(* IEC 61131-3 sources: axopen.integrations.hwc/ctrl/src (part 2) *)

                IF _progress = 452 THEN
                    TaskMessenger.ActivateOnCondition(ULINT#652, _infoTimer.output, eAxoMessageCategory#Warning);
                    IF _infoTimer.output THEN
                        Status.Error.Id := UINT#652;
                    END_IF;

                    IF TRUE THEN
                        _progress := 453;
                    END_IF;
                END_IF;

                IF _progress = 453 THEN
                    TaskMessenger.ActivateOnCondition(ULINT#653, _infoTimer.output, eAxoMessageCategory#Warning);
                    IF _infoTimer.output THEN
                        Status.Error.Id := UINT#653;
                    END_IF;

                    IF TRUE THEN
                        _progress := 454;
                    END_IF;
                END_IF;

                IF _progress = 454 THEN
                    TaskMessenger.ActivateOnCondition(ULINT#654, _infoTimer.output, eAxoMessageCategory#Warning);
                    IF _infoTimer.output THEN
                        Status.Error.Id := UINT#654;
                    END_IF;

                    IF TRUE THEN
                        _progress := 455;
                    END_IF;
                END_IF;

                IF _progress = 455 THEN
                    TaskMessenger.ActivateOnCondition(ULINT#655, _infoTimer.output, eAxoMessageCategory#Warning);
                    IF _infoTimer.output THEN
                        Status.Error.Id := UINT#655;
                    END_IF;

                    IF TRUE THEN
                        _progress := 456;
                    END_IF;
                END_IF;

                IF _progress = 456 THEN
                    TaskMessenger.ActivateOnCondition(ULINT#656, _infoTimer.output, eAxoMessageCategory#Warning);
                    IF _infoTimer.output THEN
                        Status.Error.Id := UINT#656;
                    END_IF;

                    IF TRUE THEN
                        _progress := 457;
                    END_IF;
                END_IF;

                IF _progress = 457 THEN
                    TaskMessenger.ActivateOnCondition(ULINT#657, _infoTimer.output, eAxoMessageCategory#Warning);
                    IF _infoTimer.output THEN
                        Status.Error.Id := UINT#657;
                    END_IF;

                    IF TRUE THEN
                        _progress := 458;
                    END_IF;
                END_IF;

                IF _progress = 458 THEN
                    TaskMessenger.ActivateOnCondition(ULINT#658, _infoTimer.output, eAxoMessageCategory#Warning);
                    IF _infoTimer.output THEN
                        Status.Error.Id := UINT#658;
                    END_IF;

                    IF TRUE THEN
                        _progress := 459;
                    END_IF;
                END_IF;

                IF _progress = 459 THEN
                    TemplateTask_20steps_4.DoneWhen(TRUE);
                END_IF;

                THIS.CallTimers(TRUE);

                TemplateTask_20steps_4.ThrowWhen(_errorTimer.output);
                Status.Action.Id := TO_UINT(_progress);
                TemplateTask_20steps_4.ThrowWhen(StopTask.Duration >= Config.ErrorTime ,'xxxxxxxx');
            END_IF;
            IF TemplateTask_20steps_4.DoneReached() THEN
                Status.Action.Id :=  UINT#241;
                Status.Error.Id :=  UINT#0;
            ELSIF TemplateTask_20steps_4.ErrorOccured() THEN
                Status.Action.Id :=  UINT#940;
                Status.Error.Id  :=  UINT#940;
            ELSIF TemplateTask_20steps_4.AbortTriggered()THEN
                Status.Action.Id :=  UINT#941;
                Status.Error.Id  :=  UINT#941;
            END_IF;
            Messenger.ActivateOnCondition(ULINT#940,TemplateTask_20steps_4.HasError(), eAxoMessageCategory#Error);
            Messenger.ActivateOnCondition(ULINT#941,TemplateTask_20steps_4.IsAborted(), eAxoMessageCategory#Error);
            Messenger.ActivateOnCondition(ULINT#242,TemplateTask_20steps_4.RestoreTriggered() , eAxoMessageCategory#Error);
            IF TemplateTask_20steps_4.RestoreTriggered() AND _progress >= 440 AND _progress <= 459  THEN
                Status.Action.Id :=  UINT#242;
                _progress := 0;
            END_IF;
            //******************************************

            //*************TemplateTask_20steps_5***************
            TemplateTask_20steps_5.SetIsDisabled(FALSE);
            IF TemplateTask_20steps_5.StartTriggered() THEN
                Status.Action.Id :=  UINT#260;
            END_IF;
            Messenger.ActivateOnCondition(ULINT#260,TemplateTask_20steps_5.IsBusy(), eAxoMessageCategory#Info);
            Messenger.ActivateOnCondition(ULINT#261,TemplateTask_20steps_5.IsDone(), eAxoMessageCategory#Info);
            IF TemplateTask_20steps_5.Execute() THEN
                IF _progress = 0 THEN
                    Status.Error.Id := UINT#0;
                    TaskMessenger.Restore();
                    THIS.CallTimers(FALSE);
                    _progress := 460;
                END_IF;

                IF _progress = 460 THEN
                    TaskMessenger.ActivateOnCondition(ULINT#660, _infoTimer.output, eAxoMessageCategory#Warning);
                    IF _infoTimer.output THEN
                        Status.Error.Id := UINT#660;
                    END_IF;

                    IF TRUE THEN
                        _progress := 461;
                    END_IF;
                END_IF;

                IF _progress = 461 THEN
                    TaskMessenger.ActivateOnCondition(ULINT#661, _infoTimer.output, eAxoMessageCategory#Warning);
                    IF _infoTimer.output THEN
                        Status.Error.Id := UINT#661;
                    END_IF;

                    IF TRUE THEN
                        _progress := 462;
                    END_IF;
                END_IF;

                IF _progress = 462 THEN
                    TaskMessenger.ActivateOnCondition(ULINT#662, _infoTimer.output, eAxoMessageCategory#Warning);
                    IF _infoTimer.output THEN
                        Status.Error.Id := UINT#662;
                    END_IF;

                    IF TRUE THEN
                        _progress := 463;
                    END_IF;
                END_IF;

                IF _progress = 463 THEN
                    TaskMessenger.ActivateOnCondition(ULINT#663, _infoTimer.output, eAxoMessageCategory#Warning);
                    IF _infoTimer.output THEN
                        Status.Error.Id := UINT#663;
                    END_IF;

                    IF TRUE THEN
                        _progress := 464;
                    END_IF;
                END_IF;

                IF _progress = 464 THEN
                    TaskMessenger.ActivateOnCondition(ULINT#664, _infoTimer.output, eAxoMessageCategory#Warning);
                    IF _infoTimer.output THEN
                        Status.Error.Id := UINT#664;
                    END_IF;

                    IF TRUE THEN
                        _progress := 465;
                    END_IF;
                END_IF;

                IF _progress = 465 THEN
                    TaskMessenger.ActivateOnCondition(ULINT#665, _infoTimer.output, eAxoMessageCategory#Warning);
                    IF _infoTimer.output THEN
                        Status.Error.Id := UINT#665;
                    END_IF;

                    IF TRUE THEN
                        _progress := 466;
                    END_IF;
                END_IF;

                IF _progress = 466 THEN
                    TaskMessenger.ActivateOnCondition(ULINT#666, _infoTimer.output, eAxoMessageCategory#Warning);
                    IF _infoTimer.output THEN
                        Status.Error.Id := UINT#666;
                    END_IF;

                    IF TRUE THEN
                        _progress := 467;
                    END_IF;
                END_IF;

                IF _progress = 467 THEN
                    TaskMessenger.ActivateOnCondition(ULINT#667, _infoTimer.output, eAxoMessageCategory#Warning);
                    IF _infoTimer.output THEN
                        Status.Error.Id := UINT#667;
                    END_IF;

                    IF TRUE THEN
                        _progress := 468;
                    END_IF;
                END_IF;

                IF _progress = 468 THEN
                    TaskMessenger.ActivateOnCondition(ULINT#668, _infoTimer.output, eAxoMessageCategory#Warning);
                    IF _infoTimer.output THEN
                        Status.Error.Id := UINT#668;
                    END_IF;

                    IF TRUE THEN
                        _progress := 469;
                    END_IF;
                END_IF;

                IF _progress = 469 THEN
                    TaskMessenger.ActivateOnCondition(ULINT#669, _infoTimer.output, eAxoMessageCategory#Warning);
                    IF _infoTimer.output THEN
                        Status.Error.Id := UINT#669;
                    END_IF;

                    IF TRUE THEN
                        _progress := 470;
                    END_IF;
                END_IF;

                IF _progress = 470 THEN
                    TaskMessenger.ActivateOnCondition(ULINT#670, _infoTimer.output, eAxoMessageCategory#Warning);
                    IF _infoTimer.output THEN
                        Status.Error.Id := UINT#670;
                    END_IF;

                    IF TRUE THEN
                        _progress := 471;
                    END_IF;
                END_IF;

                IF _progress = 471 THEN
                    TaskMessenger.ActivateOnCondition(ULINT#671, _infoTimer.output, eAxoMessageCategory#Warning);
                    IF _infoTimer.output THEN
                        Status.Error.Id := UINT#671;
                    END_IF;

                    IF TRUE THEN
                        _progress := 472;
                    END_IF;
                END_IF;

                IF _progress = 472 THEN
                    TaskMessenger.ActivateOnCondition(ULINT#672, _infoTimer.output, eAxoMessageCategory#Warning);
                    IF _infoTimer.output THEN
                        Status.Error.Id := UINT#672;
                    END_IF;

                    IF TRUE THEN
                        _progress := 473;
                    END_IF;
                END_IF;

                IF _progress = 473 THEN
                    TaskMessenger.ActivateOnCondition(ULINT#673, _infoTimer.output, eAxoMessageCategory#Warning);
                    IF _infoTimer.output THEN
                        Status.Error.Id := UINT#673;
                    END_IF;

                    IF TRUE THEN
                        _progress := 474;
                    END_IF;
                END_IF;

                IF _progress = 474 THEN
                    TaskMessenger.ActivateOnCondition(ULINT#674, _infoTimer.output, eAxoMessageCategory#Warning);
                    IF _infoTimer.output THEN
                        Status.Error.Id := UINT#674;
                    END_IF;

                    IF TRUE THEN
                        _progress := 475;
                    END_IF;
                END_IF;

                IF _progress = 475 THEN
                    TaskMessenger.ActivateOnCondition(ULINT#675, _infoTimer.output, eAxoMessageCategory#Warning);
                    IF _infoTimer.output THEN
                        Status.Error.Id := UINT#675;
                    END_IF;

                    IF TRUE THEN
                        _progress := 476;
                    END_IF;
                END_IF;

                IF _progress = 476 THEN
                    TaskMessenger.ActivateOnCondition(ULINT#676, _infoTimer.output, eAxoMessageCategory#Warning);
                    IF _infoTimer.output THEN
                        Status.Error.Id := UINT#676;
                    END_IF;

                    IF TRUE THEN
                        _progress := 477;
                    END_IF;
                END_IF;

                IF _progress = 477 THEN
                    TaskMessenger.ActivateOnCondition(ULINT#677, _infoTimer.output, eAxoMessageCategory#Warning);
                    IF _infoTimer.output THEN
                        Status.Error.Id := UINT#677;
                    END_IF;

                    IF TRUE THEN
                        _progress := 478;
                    END_IF;
                END_IF;

                IF _progress = 478 THEN
                    TaskMessenger.ActivateOnCondition(ULINT#678, _infoTimer.output, eAxoMessageCategory#Warning);
                    IF _infoTimer.output THEN
                        Status.Error.Id := UINT#678;
                    END_IF;

                    IF TRUE THEN
                        _progress := 479;
                    END_IF;
                END_IF;

                IF _progress = 479 THEN
                    TemplateTask_20steps_5.DoneWhen(TRUE);
                END_IF;

                THIS.CallTimers(TRUE);

                TemplateTask_20steps_5.ThrowWhen(_errorTimer.output);
                Status.Action.Id := TO_UINT(_progress);
                TemplateTask_20steps_5.ThrowWhen(StopTask.Duration >= Config.ErrorTime ,'xxxxxxxx');
            END_IF;
            IF TemplateTask_20steps_5.DoneReached() THEN
                Status.Action.Id :=  UINT#261;
                Status.Error.Id :=  UINT#0;
            ELSIF TemplateTask_20steps_5.ErrorOccured() THEN
                Status.Action.Id :=  UINT#960;
                Status.Error.Id  :=  UINT#960;
            ELSIF TemplateTask_20steps_5.AbortTriggered()THEN
                Status.Action.Id :=  UINT#961;
                Status.Error.Id  :=  UINT#961;
            END_IF;
            Messenger.ActivateOnCondition(ULINT#960,TemplateTask_20steps_5.HasError(), eAxoMessageCategory#Error);
            Messenger.ActivateOnCondition(ULINT#961,TemplateTask_20steps_5.IsAborted(), eAxoMessageCategory#Error);
            Messenger.ActivateOnCondition(ULINT#262,TemplateTask_20steps_5.RestoreTriggered() , eAxoMessageCategory#Error);
            IF TemplateTask_20steps_5.RestoreTriggered() AND _progress >= 460 AND _progress <= 479  THEN
                Status.Action.Id :=  UINT#262;
                _progress := 0;
            END_IF;
            //******************************************

        END_METHOD

        METHOD PUBLIC Stop : IAxoTaskState
            Stop := StopTask.Invoke();
        END_METHOD

        METHOD PUBLIC MoveToHome : IAxoTaskState
            MoveToHome := MoveToHomeTask.Invoke();
        END_METHOD

        METHOD PUBLIC MoveToWork : IAxoTaskState
            MoveToWork := MoveToWorkTask.Invoke();
        END_METHOD

        METHOD PROTECTED OVERRIDE ManualControl
            THIS._isManuallyControllable := true;
        END_METHOD

        ///<summary>
        /// Restores this component into intial state.
        ///</summary>
        METHOD PUBLIC OVERRIDE Restore
            Status.Action.Id :=  UINT#50;
            MoveToWorkTask.Restore();
            MoveToHomeTask.Restore();
            StopTask.Restore();

            TemplateTask_10steps_1.Restore();
            TemplateTask_10steps_2.Restore();
            TemplateTask_10steps_3.Restore();
            TemplateTask_10steps_4.Restore();
            TemplateTask_10steps_5.Restore();
            TemplateTask_20steps_1.Restore();
            TemplateTask_20steps_2.Restore();
            TemplateTask_20steps_3.Restore();
            TemplateTask_20steps_4.Restore();
            TemplateTask_20steps_5.Restore();

        END_METHOD

        METHOD PRIVATE CallTimers
            VAR_INPUT
                signal : BOOL;
            END_VAR

            _infoTimer.OnDelay(THIS, signal ,Config.InfoTime);
            _errorTimer.OnDelay(THIS, signal , Config.ErrorTime);
        END_METHOD

    END_CLASS
END_NAMESPACE

(* ---- TemplateComponent_Component_Status.st ---- *)
NAMESPACE AXOpen.Integrations.Hwc
    {S7.extern=ReadWrite}
    {#ix-attr:[Container(Layout.Stack)]}
    CLASS PUBLIC TemplateComponent_Component_Status EXTENDS AXOpen.Components.Abstractions.AxoComponent_Status
        VAR PUBLIC

        END_VAR
    END_CLASS
END_NAMESPACE

(* ---- TemplateComponent_Config.st ---- *)
NAMESPACE AXOpen.Integrations.Hwc
    {S7.extern=ReadWrite}
    {#ix-attr:[Container(Layout.Stack)]}
    CLASS PUBLIC TemplateComponent_Config
        VAR PUBLIC
            {#ix-set:AttributeName = "<#Info time#>"}
            InfoTime : LTIME := LT#5S;
            {#ix-set:AttributeName = "<#Error time#>"}
            ErrorTime : LTIME := LT#10S;
        END_VAR
    END_CLASS
END_NAMESPACE

(* ---- TemplateComponent_Control.st ---- *)
NAMESPACE AXOpen.Integrations.Hwc
    {S7.extern=ReadWrite}
    {#ix-attr:[Container(Layout.Stack)]}
    CLASS PUBLIC TemplateComponent_Control
        VAR PUBLIC
            {#ix-set:AttributeName = "<#Move home signal#>"}
            {#ix-attr:[ReadOnly()]}
            MoveHomeSignal : BOOL;
            {#ix-set:AttributeName = "<#Move work signal#>"}
            {#ix-attr:[ReadOnly()]}
            MoveWorkSignal : BOOL;
        END_VAR
    END_CLASS
END_NAMESPACE

(* ---- TemplateComponent_In.st ---- *)
NAMESPACE AXOpen.Integrations.Hwc
    {S7.extern=ReadWrite}
    {#ix-attr:[Container(Layout.Wrap)]}
    CLASS PUBLIC TemplateComponent_In
        VAR PUBLIC
            {#ix-set:AttributeName = "<#Status#>"}
            {#ix-attr:[ReadOnly()]}
            Status           :   TemplateComponent_Status;
        END_VAR
    END_CLASS
END_NAMESPACE

(* ---- TemplateComponent_Out.st ---- *)
NAMESPACE AXOpen.Integrations.Hwc
    {S7.extern=ReadWrite}
    {#ix-attr:[Container(Layout.Wrap)]}
    CLASS PUBLIC TemplateComponent_Out
        VAR PUBLIC
            {#ix-set:AttributeName = "<#Control#>"}
            {#ix-attr:[ReadOnly()]}
            Control           :   TemplateComponent_Control;
        END_VAR
    END_CLASS
END_NAMESPACE

(* ---- TemplateComponent_Status.st ---- *)
NAMESPACE AXOpen.Integrations.Hwc
    {S7.extern=ReadWrite}
    {#ix-attr:[Container(Layout.Stack)]}
    CLASS PUBLIC TemplateComponent_Status
        VAR PUBLIC
            {#ix-set:AttributeName = "<#Home sensor#>"}
            {#ix-attr:[ReadOnly()]}
            HomeSensor : BOOL;
            {#ix-set:AttributeName = "<#Work sensor#>"}
            {#ix-attr:[ReadOnly()]}
            WorkSensor : BOOL;
        END_VAR
    END_CLASS
END_NAMESPACE
